FUNCTION_BLOCK MORPHOLOGYEX (* openCV morphology ex filter *)
  (* Version 1.0, AN, SWDC RTSoft *)
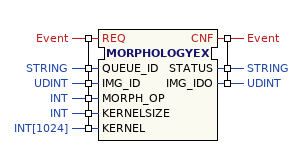
  EVENT_INPUT
    REQ WITH QUEUE_ID, IMG_ID, MORPH_OP, KERNELSIZE, KERNEL;
  END_EVENT
  EVENT_OUTPUT
    CNF WITH STATUS, IMG_IDO;
  END_EVENT
  VAR_INPUT
    QUEUE_ID : STRING;
    IMG_ID : UDINT;
    MORPH_OP : INT; (* Morphology operation: 0=ERODE, 1=DILATE, 2=OPEN, 3=CLOSE, 4=GRADIENT, 5=TOPHAT, 6=BLACKHAT *)
    KERNELSIZE : INT; (* Size of the morphology kernel. Must be a positive odd integer *)
    KERNEL : ARRAY [0..1023] OF INT; (* Morphology kernel. Array of integers will be reshaped into a square matrix *)
  END_VAR
  VAR_OUTPUT
    STATUS : STRING;
    IMG_IDO : UDINT;
  END_VAR
  ALGORITHM REQ IN ST:

  END_ALGORITHM
END_FUNCTION_BLOCK
